// Writes out part of an array of bytes.
FUNCTION F_WriteRawBytes : HRESULT
VAR_IN_OUT      
    stCtx : ST_WriteContext;
END_VAR
VAR_INPUT CONSTANT
    tBytes  : T_AnyBytes;
    nLength : UDINT;
END_VAR


F_WriteRawBytes := S_OK;

F_WriteRawBytes := F_WriteToBuffer(stCtx, tBytes, nLength);

END_FUNCTION

(* stored: Version 1.1.0.1
   POU F_WriteRawBytes: Id {03486a0e-d593-43a1-9f38-f3fba2cd9d73}, SpecialFunc None *)
